(* CODESYS project SM_MIO.library
   Description: Device support for Multi-IO 8-Layer Stackable HAT for Raspberry Pi
   Version: 1.1.0.0
   Title: Raspberry I2C MULTIIO
   Author: Sequent Microsystems
   DocFormat: reStructuredText
   Placeholder: PlaceholderTemplate
   LanguageModelAttribute: qualified-access-only
   Company: Sequent Microsystems
   DefaultNamespace: SM_MIO

Project tree, tasks and I/O mapping:
  libraries: Raspberry Pi Peripherals, 4.6.0.0 (3S - Smart Software Solutions GmbH); IoStandard, 3.5.17.0 (System); Standard, 3.5.18.0 (System)
  global variables GVL
  function block SM_MIO [ST]: AfterReadInputs, BeforeWriteOutputs
  Library Information/
    function GetLibVersionNumber [ST]
    function GetLibVersion [ST]
    function IsLibReleased [ST]
  Project Information/
    function GetCompany [ST]
    function GetTitle [ST]
    function GetVersion [ST]
    function GetTextProperty [ST]
    function GetTextProperty2 [ST]
    function GetNumberProperty [ST]
    function GetBooleanProperty [ST]
    function GetVersionProperty [ST]
  data type INT_UNION
  data type REAL_UNION
*)

// INT_UNION
TYPE INT_UNION :
UNION
	iVal: INT;
	b : ARRAY[0..1] OF BYTE;
END_UNION
END_TYPE

// REAL_UNION
TYPE REAL_UNION :
UNION
	rVal: REAL;
	b : ARRAY[0..3] OF BYTE;
END_UNION
END_TYPE

// GVL
//{attribute 'qualified_only'}
VAR_GLOBAL CONSTANT
	RELAY_VAL_ADD: USINT := 16#00;
	RELAY_SET_ADD: USINT := 16#01;
	RELAY_CLR_ADD: USINT := 16#02;
	LED_VAL_ADD: USINT := 16#03;
	OPTO_VAL_ADD: USINT := 16#06;
	U0_10_IN_VAL1_ADD: USINT := 16#08;
	I4_20_IN_VAL1_ADD: USINT := 16#0C;
	U0_10_OUT_VAL1_ADD: USINT := 16#10;
	I4_20_OUT_VAL1_ADD: USINT := 16#14;
	MOT_VAL_ADD:USINT:= 16#18;
	TEMPERATURE_ADD: USINT := 16#2E;
	SERVO_VAL1_ADD: USINT := 16#1A;
	RTD_VAL1_ADD: USINT := 16#1E;
END_VAR

// SM_MIO
FUNCTION_BLOCK SM_MIO EXTENDS i2c
VAR_INPUT
	relayState: ARRAY[0..1] OF BOOL; //-> Relays control
	ledState: ARRAY[0..5] OF BOOL; //-> Led's control
	out0_10V: ARRAY[0..1] OF REAL; //-> 0-10V output ports (V)
	out4_20mA:ARRAY[0..1] OF REAL; //-> 4 - 20mA output ports (mA)
	servo:ARRAY[0..1] OF REAL; //-> servo position [-140..140]
	motor: REAL; //-> motor pwm [0..100]
END_VAR
VAR_OUTPUT
	in0_10V: ARRAY[0..1] OF REAL; //-> 0-10V inputs ports (V)
	in4_20mA:ARRAY[0..1] OF REAL; //-> 4 - 20mA inputs ports (mA)
	inOpto: ARRAY[0..3] OF BOOL; //-> opto inputs
	inRTDTemp: ARRAY[0..1] OF REAL; //-> temperature of RTD sensors (degC)
	boardTemperature: REAL; //
END_VAR
VAR
	timer: TON := (IN:=TRUE);
	relayStateRaw: USINT;
	ledStateRaw: USINT;
	out0_10VoltRaw: ARRAY[0..1] OF UINT;
	out4_20mARaw: ARRAY[0..1] OF UINT;
	outServoRaw: ARRAY[0..1] OF INT;
	outMotorRaw: UINT;
END_VAR
VAR_TEMP	
	i, usi: USINT;
	buff: ARRAY[0..20] OF USINT;	
END_VAR

SUPER^();

CASE _iState OF
0:
	IF usiAddress < 16#06 OR  usiAddress > 16#0D THEN
		usiAddress := 16#06;
	END_IF
	
	IF SUPER^.init() THEN
		_iState := 5;
	END_IF	
5:	
	Timer.pt := T#20MS;
	buff[1] := 0;
	buff[2] := 0;
	FOR i:=0 TO 3 DO
		buff[0] := U0_10_OUT_VAL1_ADD + i* 2;
		write(ADR(buff), 3);
		out0_10VoltRaw[i] := 0;
	END_FOR
	
	// init all relay off
	
	relayStateRaw := 0;
	write8(RELAY_VAL_ADD, 0);
	
	
	_iState := 10;
END_CASE

METHOD AfterReadInputs:INT
VAR
	Buffer : ARRAY[0..3] OF BYTE;
	ch: USINT;
	address: USINT;
	value: REAL;
	len: DINT;	
	opto: USINT;
	vRUni: REAL_UNION;
END_VAR
SUPER^.AfterReadInputs();

IF _iState = 10 THEN
	timer(IN:=TRUE);
	IF timer.Q THEN	
		//opto 
		opto := read8(OPTO_VAL_ADD);  
		FOR len:=0 TO 3 DO
			inOpto[len] := USINT_TO_BOOL(SHL(2#00000001, len) AND opto);
		END_FOR
		//board temperature	
		boardTemperature := read8(TEMPERATURE_ADD);
		//RTD 
		FOR ch:=0 TO 1 DO
			address:= RTD_VAL1_ADD + 4*ch;
			len := readregister(address, ADR(Buffer), 4);		
			IF len = 4 THEN
				vRUni.b := Buffer;
				inRtdTemp[ch] := vRUni.rVal;
			END_IF
		END_FOR

		FOR ch:=0 TO 1 DO
			//0-10V inputs
			address:= U0_10_IN_VAL1_ADD + 2*ch;
			len := readregister(address, ADR(Buffer), 2);		
			IF len = 2 THEN
				value := BYTE_TO_REAL(Buffer[0]) + BYTE_TO_REAL(Buffer[1]) * 256;
				in0_10V[ch]:=value/1000;
			END_IF
			//4-20mA inputs
			address:= I4_20_IN_VAL1_ADD + 2*ch;
			len := readregister(address, ADR(Buffer), 2);		
			IF len = 2 THEN
				value := BYTE_TO_REAL(Buffer[0]) + BYTE_TO_REAL(Buffer[1]) * 256;
				in4_20mA[ch]:=value/1000;
			END_IF	
		END_FOR
		timer(IN:=FALSE);
	END_IF
END_IF
END_METHOD

METHOD BeforeWriteOutputs:INT
VAR
	i: USINT;
	cnt: USINT;
	inVal:UINT;
	inSVal:USINT;
	buff: ARRAY[0..2] OF USINT;
	wStat: BOOL;
	vIUni: INT_UNION;
END_VAR
SUPER^.BeforeWriteOutputs();

IF _iState = 10 THEN

	
	FOR i:=0 TO 1 DO
		IF out0_10V[i] < 0 THEN
			out0_10V[i] := 0;
		END_IF
		IF out0_10V[i] > 10 THEN
			out0_10V[i] := 10;
		END_IF
		IF out4_20mA[i] < 4 THEN
			out4_20mA[i] := 4;
		END_IF
		IF out4_20mA[i] > 20 THEN
			out4_20mA[i] := 20;
		END_IF
		IF servo[i] < -140 THEN
			servo[i] := -140;
		END_IF
		IF servo[i] > 140 THEN
			servo[i] := 140;
		END_IF
		// 0-10V Outputs
		inVal := REAL_TO_UINT(out0_10V[i] * 1000);
		IF out0_10VoltRaw[i] <> inVal THEN
			buff[0] := U0_10_OUT_VAL1_ADD + 2*i;
			buff[2] := UINT_TO_USINT(inVal / 256);
			buff[1] := UINT_TO_USINT(inVal - (inVal / 256));
			cnt := DINT_TO_USINT(write(ADR(buff), 3));
			IF cnt = 3 THEN
				out0_10VoltRaw[i] := inVal;
			END_IF	
		END_IF
		//4-20mA Outputs
		inVal := REAL_TO_UINT(out4_20mA[i] * 1000);
		IF out4_20mARaw[i] <> inVal THEN
			buff[0] := I4_20_OUT_VAL1_ADD + 2*i;
			buff[2] := UINT_TO_USINT(inVal / 256);
			buff[1] := UINT_TO_USINT(inVal - (inVal / 256));
			cnt := DINT_TO_USINT(write(ADR(buff), 3));
			IF cnt = 3 THEN
				out4_20mARaw[i] := inVal;
			END_IF	
		END_IF
		// servo outputs
		vIUni.iVal := REAL_TO_INT(servo[i] * 10);
		IF outServoRaw[i] <> vIUni.iVal THEN
			buff[0] := SERVO_VAL1_ADD + 2*i;
			buff[2] := vIUni.b[1];
			buff[1] := vIUni.b[0];
			cnt := DINT_TO_USINT(write(ADR(buff), 3));
			IF cnt = 3 THEN
				outServoRaw[i] := vIUni.iVal;
			END_IF	
		END_IF
	END_FOR  
	//motor
	IF motor < 0 THEN
		motor:=0;
	END_IF
	IF motor > 100 THEN
		motor:=100;
	END_IF
	inVal := REAL_TO_UINT(motor * 10);
	IF outMotorRaw <> inVal THEN
		buff[0] := MOT_VAL_ADD;
		buff[2] := UINT_TO_USINT(inVal / 256);
		buff[1] := UINT_TO_USINT(inVal - (inVal / 256));
		cnt := DINT_TO_USINT(write(ADR(buff), 3));
		IF cnt = 3 THEN
			outMotorRaw := inVal;
		END_IF	
	END_IF
	//relays
	inSVal:= 0;
	FOR i:= 0 TO 1 DO
		inSVal:= inSVal + SHL(BOOL_TO_USINT(relayState[i]), i);
	END_FOR
	IF relayStateRaw <> inSVal THEN
		IF write8(RELAY_VAL_ADD, inSVal) THEN
			relayStateRaw:=inSVal;
		END_IF
	END_IF
	//leds
	inSVal:= 0;
	FOR i:= 0 TO 5 DO
		inSVal:= inSVal + SHL(BOOL_TO_USINT(ledState[i]), i);
	END_FOR
	IF ledStateRaw <> inSVal THEN
		IF write8(LED_VAL_ADD, inSVal) THEN
			ledStateRaw:=inSVal;
		END_IF
	END_IF			
END_IF
END_METHOD

END_FUNCTION_BLOCK

// Library Information/GetLibVersionNumber
// This function has been automatically generated from the project information.
FUNCTION GetLibVersionNumber : DWORD
VAR_INPUT
	
END_VAR

GetLibVersionNumber := 16842752;

END_FUNCTION

// Project Information/GetCompany
// This function has been automatically generated from the project information.
{attribute 'signature_flag' := '1073741824'}
{attribute 'register_in_runtime'}
FUNCTION GetCompany : WSTRING
VAR_INPUT
	
END_VAR

GetCompany := "Sequent Microsystems";

END_FUNCTION

// Project Information/GetTitle
// This function has been automatically generated from the project information.
{attribute 'signature_flag' := '1073741824'}
{attribute 'register_in_runtime'}
FUNCTION GetTitle : WSTRING
VAR_INPUT
	
END_VAR

GetTitle := "Raspberry I2C MULTIIO";

END_FUNCTION

// Library Information/GetLibVersion
// This function has been automatically generated from the project information.
FUNCTION GetLibVersion : VERSION
VAR_INPUT
	
END_VAR

GetLibVersion.uiMajor := 1;
GetLibVersion.uiMinor := 1;
GetLibVersion.uiServicePack := 0;
GetLibVersion.uiPatch := 0;

END_FUNCTION

// Library Information/IsLibReleased
// This function has been automatically generated from the project information.
FUNCTION IsLibReleased : BOOL
VAR_INPUT
	
END_VAR

IsLibReleased := FALSE;

END_FUNCTION

// Project Information/GetVersion
// This function has been automatically generated from the project information.
{attribute 'signature_flag' := '1073741824'}
{attribute 'register_in_runtime'}
FUNCTION GetVersion : VERSION
VAR_INPUT
	
END_VAR

GetVersion.uiMajor := 1;
GetVersion.uiMinor := 1;
GetVersion.uiServicePack := 0;
GetVersion.uiPatch := 0;

END_FUNCTION

// Project Information/GetTextProperty
// This function has been automatically generated from the project information.
{attribute 'signature_flag' := '1073741824'}
{attribute 'register_in_runtime'}
FUNCTION GetTextProperty : WSTRING
VAR_INPUT
	stKey: WSTRING;
END_VAR

IF stKey = "Author" THEN
	GetTextProperty := "Sequent Microsystems";
ELSIF stKey = "Company" THEN
	GetTextProperty := "Sequent Microsystems";
ELSIF stKey = "DefaultNamespace" THEN
	GetTextProperty := "SM_MIO";
ELSIF stKey = "Description" THEN
	GetTextProperty := "Device support for Multi-IO 8-Layer Stackable HAT for Raspberry Pi";
ELSIF stKey = "DocFormat" THEN
	GetTextProperty := "reStructuredText";
ELSIF stKey = "LanguageModelAttribute" THEN
	GetTextProperty := "qualified-access-only";
ELSIF stKey = "Placeholder" THEN
	GetTextProperty := "PlaceholderTemplate";
ELSIF stKey = "Project" THEN
	GetTextProperty := "SM_MIO";
ELSIF stKey = "Title" THEN
	GetTextProperty := "Raspberry I2C MULTIIO";
ELSE
	GetTextProperty := "";
END_IF

END_FUNCTION

// Project Information/GetTextProperty2
// This function has been automatically generated from the project information.
{attribute 'signature_flag' := '1073741824'}
{attribute 'register_in_runtime'}
FUNCTION GetTextProperty2 : POINTER TO WSTRING
VAR_INPUT
	stKey: WSTRING;
END_VAR

IF stKey = "Author" THEN
	GetTextProperty2 := ADR("Sequent Microsystems");
ELSIF stKey = "Company" THEN
	GetTextProperty2 := ADR("Sequent Microsystems");
ELSIF stKey = "DefaultNamespace" THEN
	GetTextProperty2 := ADR("SM_MIO");
ELSIF stKey = "Description" THEN
	GetTextProperty2 := ADR("Device support for Multi-IO 8-Layer Stackable HAT for Raspberry Pi");
ELSIF stKey = "DocFormat" THEN
	GetTextProperty2 := ADR("reStructuredText");
ELSIF stKey = "LanguageModelAttribute" THEN
	GetTextProperty2 := ADR("qualified-access-only");
ELSIF stKey = "Placeholder" THEN
	GetTextProperty2 := ADR("PlaceholderTemplate");
ELSIF stKey = "Project" THEN
	GetTextProperty2 := ADR("SM_MIO");
ELSIF stKey = "Title" THEN
	GetTextProperty2 := ADR("Raspberry I2C MULTIIO");
ELSE
	GetTextProperty2 := ADR("");
END_IF

END_FUNCTION

// Project Information/GetNumberProperty
// This function has been automatically generated from the project information.
{attribute 'signature_flag' := '1073741824'}
{attribute 'register_in_runtime'}
FUNCTION GetNumberProperty : DINT
VAR_INPUT
	stKey: WSTRING;
END_VAR

GetNumberProperty := 0;

END_FUNCTION

// Project Information/GetBooleanProperty
// This function has been automatically generated from the project information.
{attribute 'signature_flag' := '1073741824'}
{attribute 'register_in_runtime'}
FUNCTION GetBooleanProperty : BOOL
VAR_INPUT
	stKey: WSTRING;
END_VAR

IF stKey = "IsEndUserLibrary" THEN
	GetBooleanProperty := FALSE;
ELSIF stKey = "Released" THEN
	GetBooleanProperty := FALSE;
ELSE
	GetBooleanProperty := FALSE;
END_IF

END_FUNCTION

// Project Information/GetVersionProperty
// This function has been automatically generated from the project information.
{attribute 'signature_flag' := '1073741824'}
{attribute 'register_in_runtime'}
FUNCTION GetVersionProperty : VERSION
VAR_INPUT
	stKey: WSTRING;
END_VAR

IF stKey = "Version" THEN
	GetVersionProperty.uiMajor := 1;
	GetVersionProperty.uiMinor := 1;
	GetVersionProperty.uiServicePack := 0;
	GetVersionProperty.uiPatch := 0;
ELSE
	GetVersionProperty.uiMajor := 0;
	GetVersionProperty.uiMinor := 0;
	GetVersionProperty.uiServicePack := 0;
	GetVersionProperty.uiPatch := 0;
END_IF

END_FUNCTION
